Universal Robots URScript: Test Teach Position Straight.script

def Test_Teach_Position_Straight():
  global _hidden_verificationVariable=0
  set_standard_analog_input_domain(0, 1)
  set_standard_analog_input_domain(1, 1)
  set_tool_analog_input_domain(0, 1)
  set_tool_analog_input_domain(1, 1)
  set_analog_outputdomain(0, 0)
  set_analog_outputdomain(1, 0)
  set_input_actions_to_default()
  set_safety_mode_transition_hardness(1)
  set_target_payload(10.800000, [-0.001000, -0.053000, 0.068000], [0.081228, 0.081228, 0.081228, 0.000000, 0.000000, 0.000000])
  set_tool_communication(False, 115200, 0, 1, 1.5, 3.5)
  set_tool_output_mode(0)
  set_tool_digital_output_mode(0, 1)
  set_tool_digital_output_mode(1, 1)
  set_tool_voltage(0)
  set_tcp(p[-0.0095,-0.328,0.10573,1.2092,-1.2092,1.2092])
  set_gravity([0.0, 0.0, 9.82])
  global robot_number=2
  global Point_1=p[0.0,0.0,0.0,0.0,0.0,0.0]
  global Point_2=p[0.0,0.0,0.0,0.0,0.0,0.0]
  # begin: URCap Installation Node
  #   Source: UR Connect, 1.13.79, Universal Robots
  #   Type: UR Connect
  myurRPC = rpc_factory("xmlrpc","http://127.0.0.1:40474")
  # end: URCap Installation Node
  # begin: URCap Installation Node
  #   Source: MachineLogic for Universal Robots, 3.1.7, Vention Inc.
  #   Type: MachineLogic for Universal Robots
  def waitForResponse(expected_response_vention, cname_vention):
  response_vention = socket_read_string(cname_vention,timeout=15)
  while response_vention != expected_response_vention:
  sleep(0.01)
  response_vention = socket_read_string(cname_vention,timeout=15)
  end
  sleep(0.01)
  sync()
  end
  def sendString(string_vention, expected_response_vention, cname_vention):
  socket_send_string(str_cat(string_vention,";"), cname_vention)
  response_vention = socket_read_string(cname_vention,timeout=15)
  if(response_vention == "nAck"):
  popup("nAck received")
  end
  while response_vention != expected_response_vention:
  sleep(0.01)
  response_vention = socket_read_string(cname_vention,timeout=15)
  if(response_vention == "nAck"):
  popup("nAck received")
  end
  end
  sleep(0.01)
  sync()
  end
  def sendStringNAck(string_vention, expected_response_vention, cname_vention):
  socket_send_string(str_cat(string_vention,";"), cname_vention)
  response_vention = socket_read_string(cname_vention,timeout=15)
  if(response_vention == "nAck"):
  popup("nAck received")
  end
  while(response_vention != expected_response_vention and response_vention != "nAck"):
  sleep(0.01)
  response_vention = socket_read_string(cname_vention,timeout=15)
  if(response_vention == "nAck"):
  popup("nAck received",blocking=True)
  end
  end
  sleep(0.01)
  sync()
  end
  def sendStringWithTimeout(string_vention, expected_response_vention, cname_vention):
  socket_send_string(str_cat(string_vention,";"), cname_vention)
  response_vention = socket_read_string(cname_vention,timeout=10)
  if(response_vention == "nAck"):
  popup("nAck received"+string_vention)
  end
  sleep(0.01)
  sync()
  end
  def pollString(string_vention, expected_response_vention, cname_vention):
  socket_send_string(str_cat(string_vention,";"), cname_vention)
  response_vention = socket_read_string(cname_vention,timeout=15)
  if(response_vention == "nAck"):
  popup("nAck received")
  end
  while response_vention != expected_response_vention:
  sleep(1)
  socket_send_string(str_cat(string_vention,";"), cname_vention)
  response_vention = socket_read_string(cname_vention,timeout=15)
  if(response_vention == "nAck"):
  popup("nAck received")
  end
  end
  sleep(0.01)
  sync()
  end
  def sendVariable(var_vention, data_vention, expected_response_vention, cname_vention):
  socket_set_var(var_vention, data_vention, cname_vention)
  response_vention = socket_read_string(cname_vention,timeout=15)
  if(response_vention == "nAck"):
  popup("nAck received")
  end
  while response_vention != expected_response_vention:
  sleep(0.01)
  response_vention = socket_read_string(cname_vention,timeout=15)
  if(response_vention == "nAck"):
  popup("nAck received")
  end
  end
  sleep(0.01)
  sync()
  end
  def intToString(integer_vention,cname_vention):
  stringFix=""
  multiplier_vention123=1
  if integer_vention<0:
  stringFix="-"
  multiplier_vention123=-1
  end
  socket_set_var("GetString",integer_vention*multiplier_vention123,cname_vention)
  string_vention=""
  while string_vention=="":
  sleep(0.01)
  string_vention=socket_read_string(cname_vention,timeout=15)
  end
  sleep(0.01)
  sync()
  string_vention=stringFix+string_vention
  return string_vention
  end
  string_vention=""
  isVentionMovementBusy = False
  isVentionParallelMovementSendingScript = False
  ventionThreadHandle = 1
  isVentionMovementBusyMachineMotion1 = False
  isVentionParallelMovementSendingScriptMachineMotion1 = False
  socket_vention = socket_open("192.168.3.52", 9999, "MachineMotion1")
  if socket_vention==False:
  popup("Check configuration, can't connect to MachineMotion")
  end
  waitForResponse("MachineMotion connection established", "MachineMotion1")
  sendString("isReady", "MachineMotion isReady = true", "MachineMotion1")
  sendStringWithTimeout("setURCapVersion2", "setURCapVersion loaded", "MachineMotion1")
  sendString("SET speed_v2 1000000", "Ack", "MachineMotion1")
  sendString("SET acceleration_v2 100000", "Ack", "MachineMotion1")
  sendString("SET de_axis_1_microsteps_config 8", "Ack", "MachineMotion1")
  sendString("SET de_axis_1_mechanical_gain_config_v2 150000.0", "Ack", "MachineMotion1")
  sendString("SET de_axis_1_direction_config 1", "Ack", "MachineMotion1")
  sendString("SET de_axis_1_type_config Custom Actuator ", "Ack", "MachineMotion1")
  sendString("de_axis_1_config_exec", "Ack", "MachineMotion1")
  # end: URCap Installation Node
  # begin: URCap Installation Node
  #   Source: WireTank Serial, 4.9.0, WireTank, LLC
  #   Type: WireTank Serial
  WTSerialBridge = rpc_factory("xmlrpc","http://127.0.0.1:40511/RPC2")
  # end: URCap Installation Node
  step_count_935dbc96_cd99_4121_ab5b_d3d6ef4dec80 = 0.0
  thread Step_Counter_Thread_73284af6_db75_4028_af7c_79f71c37ba19():
    while (True):
      step_count_935dbc96_cd99_4121_ab5b_d3d6ef4dec80 = step_count_935dbc96_cd99_4121_ab5b_d3d6ef4dec80 + 1.0
      sync()
    end
  end
  run Step_Counter_Thread_73284af6_db75_4028_af7c_79f71c37ba19()
  global freedrive_m_var=  False
  global Waypoint_40_p=p[.360688403366, .270119715397, .646144746546, .057805349154, 2.125995180379, 2.134053153683]
  global Waypoint_40_q=[-3.4579489866839808, -2.0569035015501917, 2.3265796343432825, -0.22706706941638188, -0.1993501822101038, -0.10534793535341436]
  global Waypoint_2_p=p[-.548957282596, .386284559177, .143710178207, 1.570800598292, -.000025190822, .000004803470]
  global Waypoint_2_q=[-1.0516188780414026, -1.010990933781006, 2.1562450567828577, -1.143702046280243, -1.0526168982135218, -0.0017235914813440445]
  while (True):
    $ 2 "Robot Program"
    $ 6 "MoveJ"
    $ 7 "Waypoint_40" "breakAfter"
    set_tcp(p[0.0,0.0,0.019,0.0,0.0,0.0])
    movej(get_inverse_kin(Waypoint_40_p, qnear=Waypoint_40_q), a=1.3962634015954636, v=1.0471975511965976)
    $ 8 "'above waypoint is home'"
    # 'above waypoint is home'
    $ 9 "Waypoint_2" "breakAfter"
    set_tcp(p[0.0,0.0,0.019,0.0,0.0,0.0])
    movej(get_inverse_kin(Waypoint_2_p, qnear=Waypoint_2_q), a=1.3962634015954636, v=1.0471975511965976)
    $ 10 "freedrive_m_var≔ False "
    global freedrive_m_var=  False
    $ 11 "freedrive_m_var≔ True "
    global freedrive_m_var=  True
    $ 12 "Popup: Move the TCP to the left side of the weld (very end of the V chisel), then click 'Continue'"
    popup("Move the TCP to the left side of the weld (very end of the V chisel), then click 'Continue'", "Message", False, False, blocking=True)
    $ 13 "tcp_pose_left≔get_actual_tcp_pose()"
    global tcp_pose_left= get_actual_tcp_pose ()
    $ 14 "Popup: Move the TCP to the right side of the weld (very end of the V chisel), then click 'Continue'"
    popup("Move the TCP to the right side of the weld (very end of the V chisel), then click 'Continue'", "Message", False, False, blocking=True)
    $ 15 "tcp_pose_right≔get_actual_tcp_pose()"
    global tcp_pose_right= get_actual_tcp_pose ()
    $ 16 "freedrive_m_var≔ False "
    global freedrive_m_var=  False
    $ 17 "Wait: 0.25"
    sleep(0.25)
    $ 18 "sync()"
    sync()
  end
end
